# EPICS substitutions: db/Beckhoff_5XXX/ecmcEL5021.substitutions
file "ecmcEcSlave.template"
{
  pattern {}
          {}
}

# All fields related to postion scaling and alarms
file "ecmcEL5021-chX.template"
{
  pattern {CH_ID}
          {01   }
}
